FUNCTION_BLOCK AUS_SPLIT_8 (* SPLIT 1 AUS into 8 AUS (generic FB) *)
  (* Standard: 61499-2; Description: Copyright (c) 2025 HR Agrartechnik GmbH This program and the accompanying materials are made available under the terms of the Eclipse Public License 2.0 which is available at https://www.eclipse.org/legal/epl-2.0/ SPDX-License-Identifier: EPL-2.0 *)
  (* Version 1.0, 2025-01-24, Franz Höpfinger, HR Agrartechnik GmbH *)
  PACKAGE adapter::events::unidirectional;
  IMPORT eclipse4diac::core::GenericClassName;
  {SET_ATTRIBUTE(eclipse4diac::core::GenericClassName, 'GEN_AUS_SPLIT')}
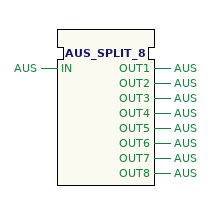
  SOCKETS
    IN : adapter::types::unidirectional::AUS;
  END_SOCKETS
  PLUGS
    OUT1 : adapter::types::unidirectional::AUS;
    OUT2 : adapter::types::unidirectional::AUS;
    OUT3 : adapter::types::unidirectional::AUS;
    OUT4 : adapter::types::unidirectional::AUS;
    OUT5 : adapter::types::unidirectional::AUS;
    OUT6 : adapter::types::unidirectional::AUS;
    OUT7 : adapter::types::unidirectional::AUS;
    OUT8 : adapter::types::unidirectional::AUS;
  END_PLUGS
END_FUNCTION_BLOCK
